VAR_GLOBAL // TIMERS
    timer0: TON;
    timer1: TON;
    curTimer: INT := 0;
END_VAR

(* stored: ProductVersion 3.1.0.18, Version 1.1.0.1 *)
